FUNCTION F_ComputeSFixed32Size : UDINT
VAR_INPUT
    {attribute 'analysis' := '-33' }
    nValue : DINT;
END_VAR


F_ComputeSFixed32Size := GCL_PB.cLittleEndian32Size;

END_FUNCTION

(* stored: Version 1.1.0.1
   POU F_ComputeSFixed32Size: Id {b2117b92-1980-4b3f-ade2-c2136604f85c}, SpecialFunc None *)
